// TIA Portal V20 export
// export: Created 2025-12-01T14:57:06.2911108Z, ExportSetting None, DisplayName Totally Integrated Automation Portal, DisplayVersion V20 Update 3, DisplayName TIA Portal Openness, DisplayVersion V20 Update 3, DisplayName TIA Portal Version Control Interface, DisplayVersion V20 Update 3, DisplayName STEP 7 Professional, DisplayVersion V20 Update 3, DisplayName STEP 7 Safety, DisplayVersion V20 Update 2, DisplayName WinCC Basic/Comfort/Advanced, DisplayVersion V20 Update 3, DisplayName WinCC Professional, DisplayVersion V20 Update 3, DisplayName WinCC Unified, DisplayVersion V20 Update 3
FUNCTION "FC912_CNT_Tiempo_Mem_UHS" : Void   // FC912, LAD
{ S7_Optimized_Access := 'FALSE' }
AUTHOR : GENERAL
NAME : 20130301
VERSION : 3.0
// stored: AutoNumber false, SetENOAutomatically false
   VAR_INPUT
      Temporizar : Bool;
      Reset : Bool;
      Valor_Tiempo : UDInt;
      Base_tiempo_ms : UDInt;
   END_VAR
   VAR_OUTPUT
      Tiempo_OK : Bool;
   END_VAR
   VAR_IN_OUT
      Valor_Actual : UDInt;
   END_VAR
   VAR_TEMP
      Aux_Inc_Tiempo : UDInt;
      TEMP_Tiempo_OK : Bool;
   END_VAR
BEGIN

REGION Network 1: ---
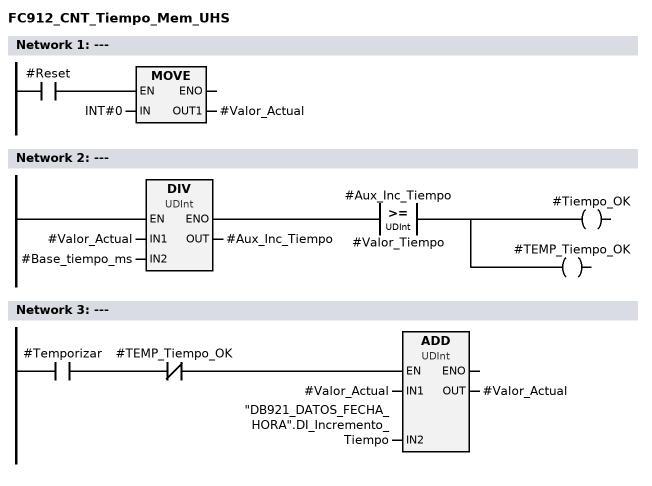
   RUNG wire#powerrail
      Contact( #Reset )
      { S7_GenerateENO := "TRUE" } Move(in := INT#0, out1 => #Valor_Actual)
   END_RUNG
   // the same network as SCL:
   IF #Reset THEN #Valor_Actual := INT#0; END_IF;
END_REGION

REGION Network 2: ---
   RUNG wire#powerrail
      { S7_Templates := "SrcType := UDInt"; S7_GenerateENO := "TRUE" } Div(in1 := #Valor_Actual, in2 := #Base_tiempo_ms, out => #Aux_Inc_Tiempo)
      { S7_Templates := "SrcType := UDInt" } GE_Contact(in1 := #Aux_Inc_Tiempo, in2 := #Valor_Tiempo)
      wire#w1
      Coil( #Tiempo_OK )
   END_RUNG
   RUNG wire#w1
      Coil( #TEMP_Tiempo_OK )
   END_RUNG
   // the same network as SCL:
   // ENO of a box is taken as its EN; it also drops when the box reports an error
   #Aux_Inc_Tiempo := #Valor_Actual / #Base_tiempo_ms;
   #Tiempo_OK := #Aux_Inc_Tiempo >= #Valor_Tiempo;
   #TEMP_Tiempo_OK := #Tiempo_OK;
END_REGION

REGION Network 3: ---
   RUNG wire#powerrail
      Contact( #Temporizar )
      I_Contact( #TEMP_Tiempo_OK )
      { S7_Templates := "SrcType := UDInt"; S7_GenerateENO := "TRUE" } Add(in1 := #Valor_Actual, in2 := "DB921_DATOS_FECHA_HORA".DI_Incremento_Tiempo, out => #Valor_Actual)
   END_RUNG
   // the same network as SCL:
   IF #Temporizar AND NOT #TEMP_Tiempo_OK THEN
       #Valor_Actual := #Valor_Actual + "DB921_DATOS_FECHA_HORA".DI_Incremento_Tiempo;
   END_IF;
END_REGION
END_FUNCTION
